// TIA Portal V17 export
// export: Created 2023-04-11T09:33:28.0582979Z, ExportSetting WithDefaults, DisplayName Totally Integrated Automation Portal, DisplayVersion V17 Update 3, DisplayName TIA Portal Openness, DisplayVersion V17 Update 3, DisplayName TIA Portal Version Control Interface, DisplayVersion V17, DisplayName SINAMICS Startdrive Advanced, DisplayVersion V17 Update2, DisplayName SINAMICS Startdrive G130, G150, S120, S150, SINAMICS MV, S210, DisplayVersion V17 Update2, DisplayName SINAMICS Startdrive G110M, G120, G120C, G120D, G120P, G115D, DisplayVersion V17 Update2, DisplayName STEP 7 Professional, DisplayVersion V17 Update 3, DisplayName STEP 7 Safety, DisplayVersion V17, DisplayName WinCC UA Professional, DisplayVersion V17 Update 3
FUNCTION_BLOCK "FB_stdStep"   // FB113, LAD
{ S7_Optimized_Access := 'TRUE' }
VERSION : 0.1
// Standard program step
// stored: AutoNumber true, IsIECCheckEnabled false, IsRetainMemResEnabled false, MemoryReserve 100, SetENOAutomatically false, UDAEnableTagReadback false
   VAR_INPUT
      enable { ExternalAccessible := 'False'; ExternalVisible := 'False'; ExternalWritable := 'False'} : Bool;
      condition { ExternalAccessible := 'False'; ExternalVisible := 'False'; ExternalWritable := 'False'} : Bool;
      delay { ExternalAccessible := 'False'; ExternalVisible := 'False'; ExternalWritable := 'False'} : Time;
      timeout { ExternalAccessible := 'False'; ExternalVisible := 'False'; ExternalWritable := 'False'} : Time;
   END_VAR
   VAR_OUTPUT
      done { ExternalAccessible := 'False'; ExternalVisible := 'False'; ExternalWritable := 'False'} : Bool;
      error { ExternalAccessible := 'False'; ExternalVisible := 'False'; ExternalWritable := 'False'} : Bool;
      out { ExternalAccessible := 'False'; ExternalVisible := 'False'; ExternalWritable := 'False'} : Bool;
      out_pls { ExternalAccessible := 'False'; ExternalVisible := 'False'; ExternalWritable := 'False'} : Bool;
      out_plf { ExternalAccessible := 'False'; ExternalVisible := 'False'; ExternalWritable := 'False'} : Bool;
   END_VAR
   VAR
      temp_1 { ExternalAccessible := 'False'; ExternalVisible := 'False'; ExternalWritable := 'False'} : Bool;
      temp_2 { ExternalAccessible := 'False'; ExternalVisible := 'False'; ExternalWritable := 'False'} : Bool;
      IEC_Timer_Instance_1 { ExternalAccessible := 'False'; ExternalVisible := 'False'; ExternalWritable := 'False'; S7_SetPoint := 'True'} : TON_TIME;
      IEC_Timer_Instance_2 { ExternalAccessible := 'False'; ExternalVisible := 'False'; ExternalWritable := 'False'; S7_SetPoint := 'True'} : TON_TIME;
   END_VAR
   VAR_TEMP   // added for the SCL form of the ladder/FBD networks
      _w1 : Bool;
      _w2 : Bool;
   END_VAR
BEGIN

REGION Network 1: Done and Error output logic
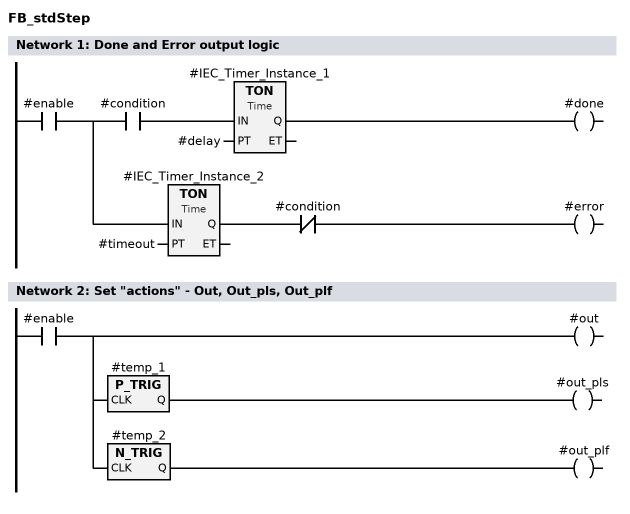
   RUNG wire#powerrail
      Contact( #enable )
      wire#w1
      Contact( #condition )
      { S7_Templates := "time_type := Time" } #IEC_Timer_Instance_1.TON(pt := #delay, et =>)
      Coil( #done )
   END_RUNG
   RUNG wire#w1
      { S7_Templates := "time_type := Time" } #IEC_Timer_Instance_2.TON(pt := #timeout, et =>)
      I_Contact( #condition )
      Coil( #error )
   END_RUNG
   // the same network as SCL:
   #IEC_Timer_Instance_1(IN := #enable AND #condition, PT := #delay);   // TON
   #done := #IEC_Timer_Instance_1.Q;
   #IEC_Timer_Instance_2(IN := #enable, PT := #timeout);   // TON
   #error := #IEC_Timer_Instance_2.Q AND NOT #condition;
END_REGION

REGION Network 2: Set "actions" - Out, Out_pls, Out_plf
   RUNG wire#powerrail
      Contact( #enable )
      wire#w1
      Coil( #out )
   END_RUNG
   RUNG wire#w1
      P_Trig( #temp_1 )
      Coil( #out_pls )
   END_RUNG
   RUNG wire#w1
      N_Trig( #temp_2 )
      Coil( #out_plf )
   END_RUNG
   // the same network as SCL:
   #out := #enable;
   #_w1 := #enable AND NOT #temp_1;   // rising edge
   #temp_1 := #enable;
   #out_pls := #_w1;
   #_w2 := NOT #enable AND #temp_2;   // falling edge
   #temp_2 := #enable;
   #out_plf := #_w2;
END_REGION
END_FUNCTION_BLOCK
